// TIA Portal V20 export
FUNCTION "Service_Dosing" : Void   // FC11, FBD
TITLE = Service
{ S7_Optimized_Access := 'TRUE' }
AUTHOR : Siemens AG
FAMILY : ServiceControl
VERSION : 1.0
// stored: SetENOAutomatically false
   VAR_TEMP
      State : "Service_States";
   END_VAR
BEGIN

REGION Network 1: Cm P100 feedback
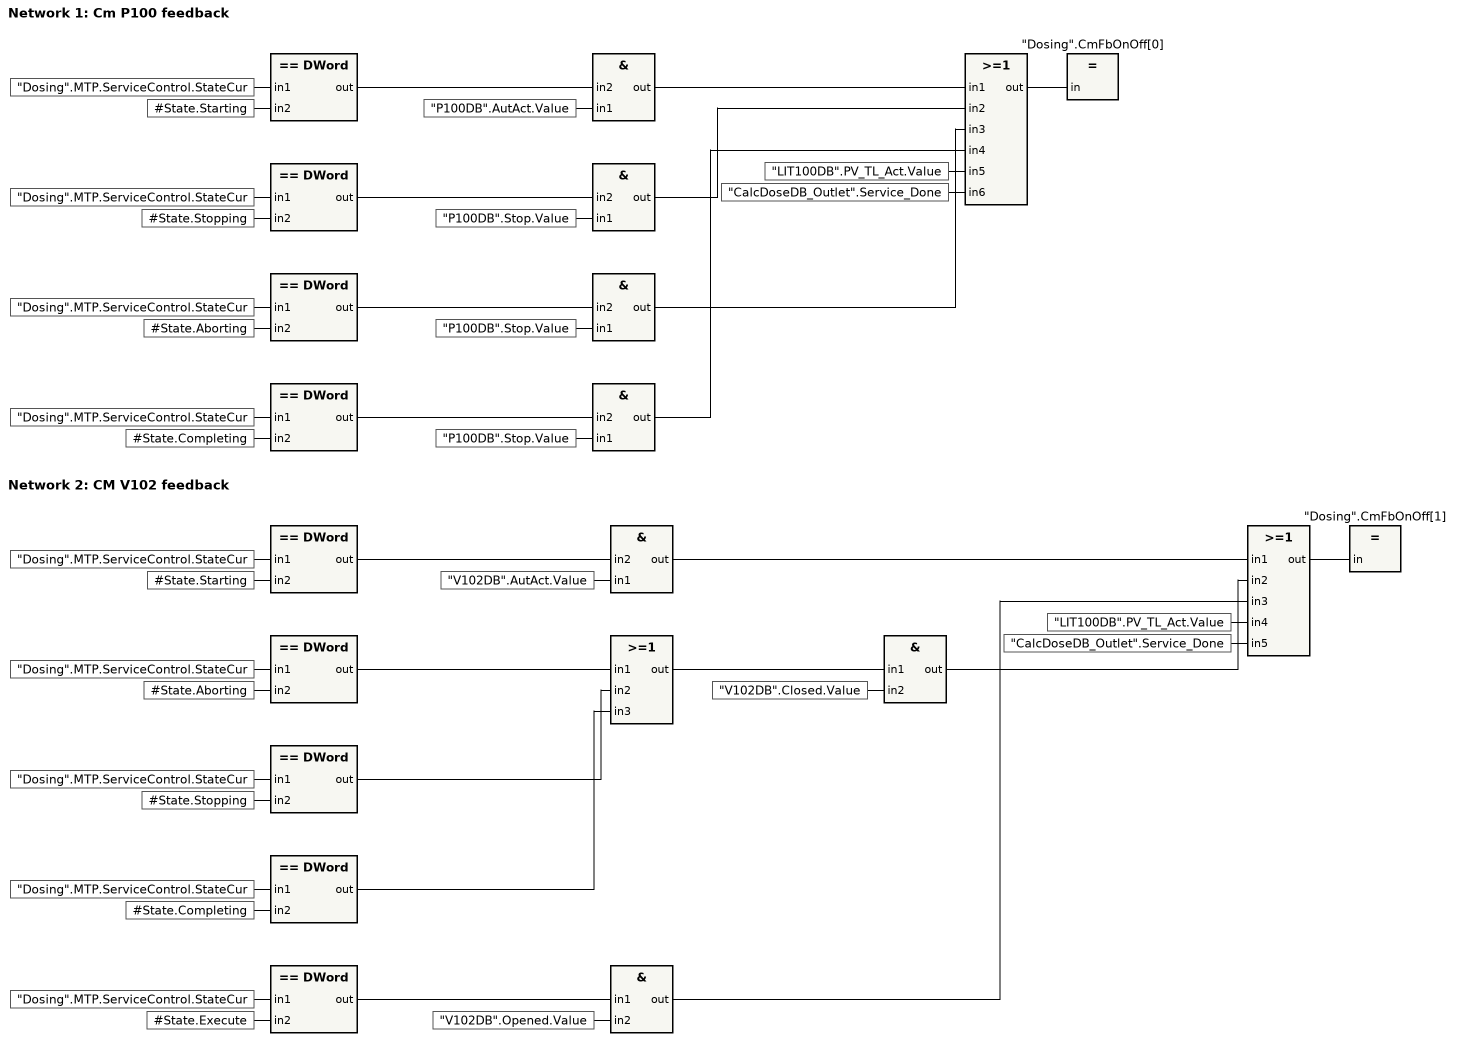
   "Dosing".CmFbOnOff[0] := (("Dosing".MTP.ServiceControl.StateCur = #State.Starting) AND "P100DB".AutAct.Value) OR (("Dosing".MTP.ServiceControl.StateCur = #State.Stopping) AND "P100DB".Stop.Value) OR (("Dosing".MTP.ServiceControl.StateCur = #State.Aborting) AND "P100DB".Stop.Value) OR (("Dosing".MTP.ServiceControl.StateCur = #State.Completing) AND "P100DB".Stop.Value) OR "LIT100DB".PV_TL_Act.Value OR "CalcDoseDB_Outlet".Service_Done;
END_REGION

REGION Network 2: CM V102 feedback
   "Dosing".CmFbOnOff[1] := (("Dosing".MTP.ServiceControl.StateCur = #State.Starting) AND "V102DB".AutAct.Value) OR ((("Dosing".MTP.ServiceControl.StateCur = #State.Aborting) OR ("Dosing".MTP.ServiceControl.StateCur = #State.Stopping) OR ("Dosing".MTP.ServiceControl.StateCur = #State.Completing)) AND "V102DB".Closed.Value) OR (("Dosing".MTP.ServiceControl.StateCur = #State.Execute) AND "V102DB".Opened.Value) OR "LIT100DB".PV_TL_Act.Value OR "CalcDoseDB_Outlet".Service_Done;
END_REGION

REGION Network 3: CM V103 feedback
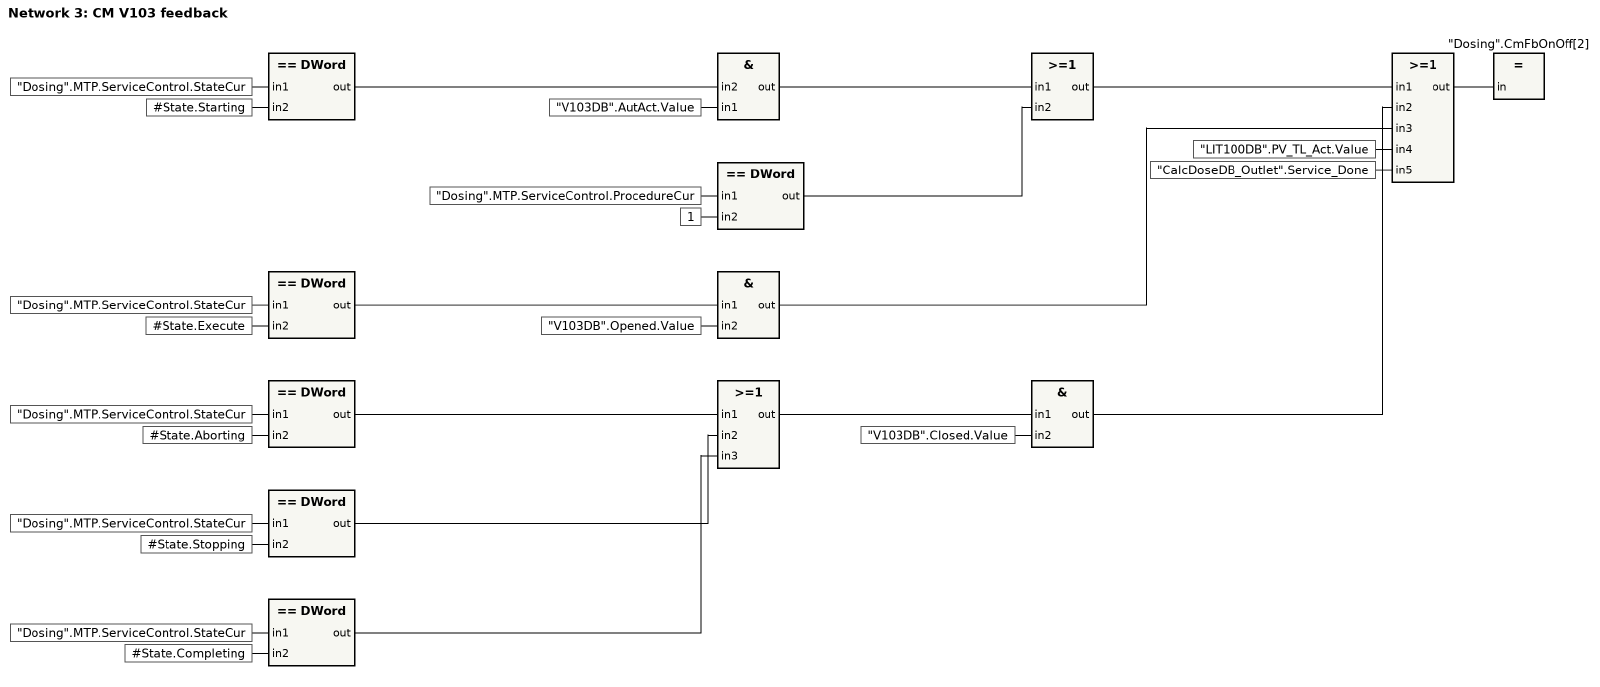
   "Dosing".CmFbOnOff[2] := (("Dosing".MTP.ServiceControl.StateCur = #State.Starting) AND "V103DB".AutAct.Value) OR ("Dosing".MTP.ServiceControl.ProcedureCur = 1) OR ((("Dosing".MTP.ServiceControl.StateCur = #State.Aborting) OR ("Dosing".MTP.ServiceControl.StateCur = #State.Stopping) OR ("Dosing".MTP.ServiceControl.StateCur = #State.Completing)) AND "V103DB".Closed.Value) OR (("Dosing".MTP.ServiceControl.StateCur = #State.Execute) AND "V103DB".Opened.Value) OR "LIT100DB".PV_TL_Act.Value OR "CalcDoseDB_Outlet".Service_Done;
END_REGION

REGION Network 4: CM V104 feedback
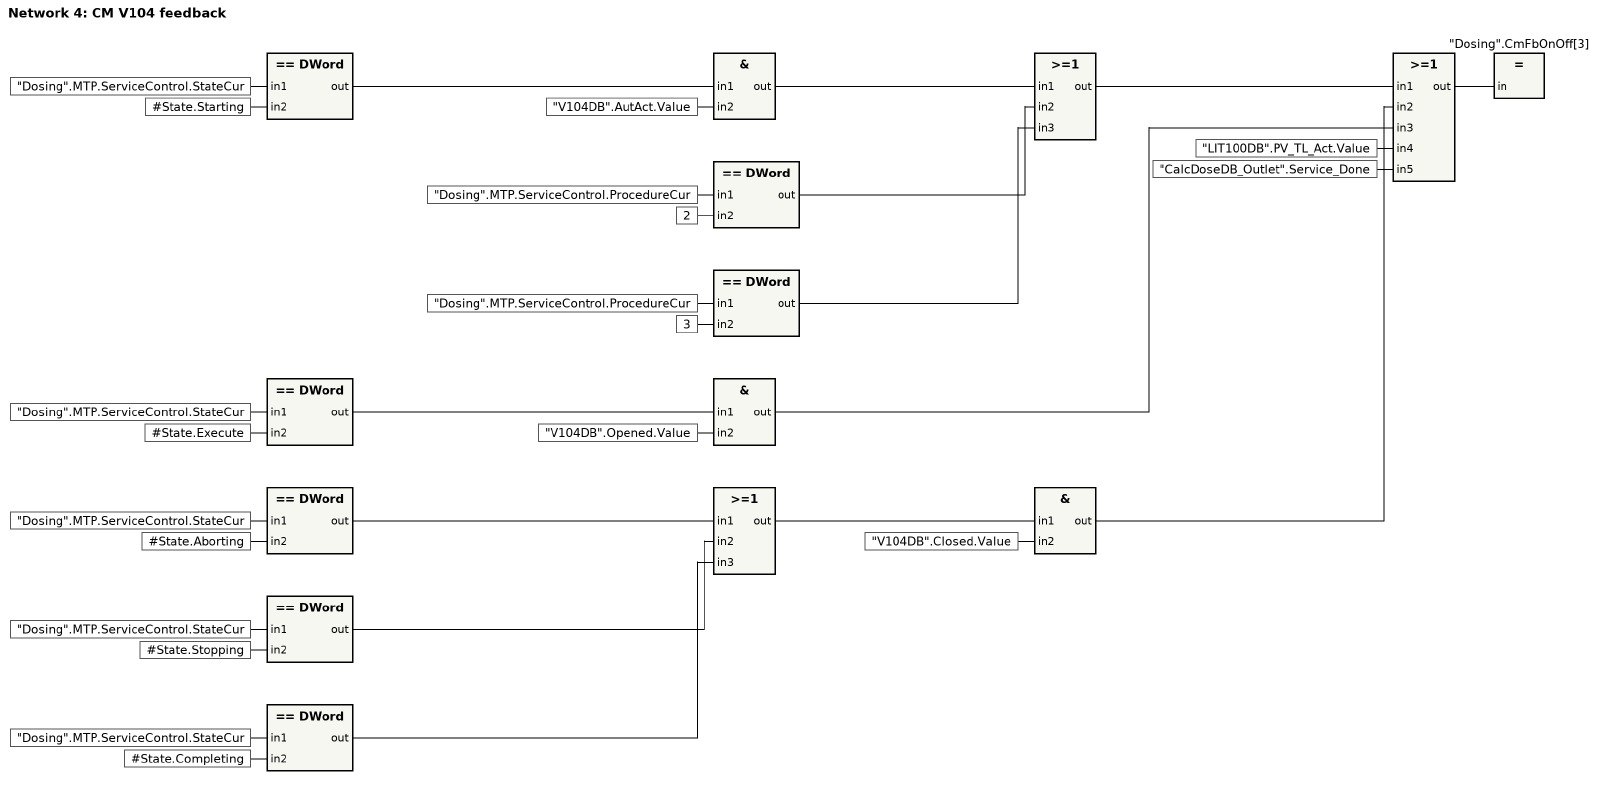
   "Dosing".CmFbOnOff[3] := (("Dosing".MTP.ServiceControl.StateCur = #State.Starting) AND "V104DB".AutAct.Value) OR ("Dosing".MTP.ServiceControl.ProcedureCur = 2) OR ("Dosing".MTP.ServiceControl.ProcedureCur = 3) OR ((("Dosing".MTP.ServiceControl.StateCur = #State.Aborting) OR ("Dosing".MTP.ServiceControl.StateCur = #State.Stopping) OR ("Dosing".MTP.ServiceControl.StateCur = #State.Completing)) AND "V104DB".Closed.Value) OR (("Dosing".MTP.ServiceControl.StateCur = #State.Execute) AND "V104DB".Opened.Value) OR "LIT100DB".PV_TL_Act.Value OR "CalcDoseDB_Outlet".Service_Done;
END_REGION

REGION Network 5: Service
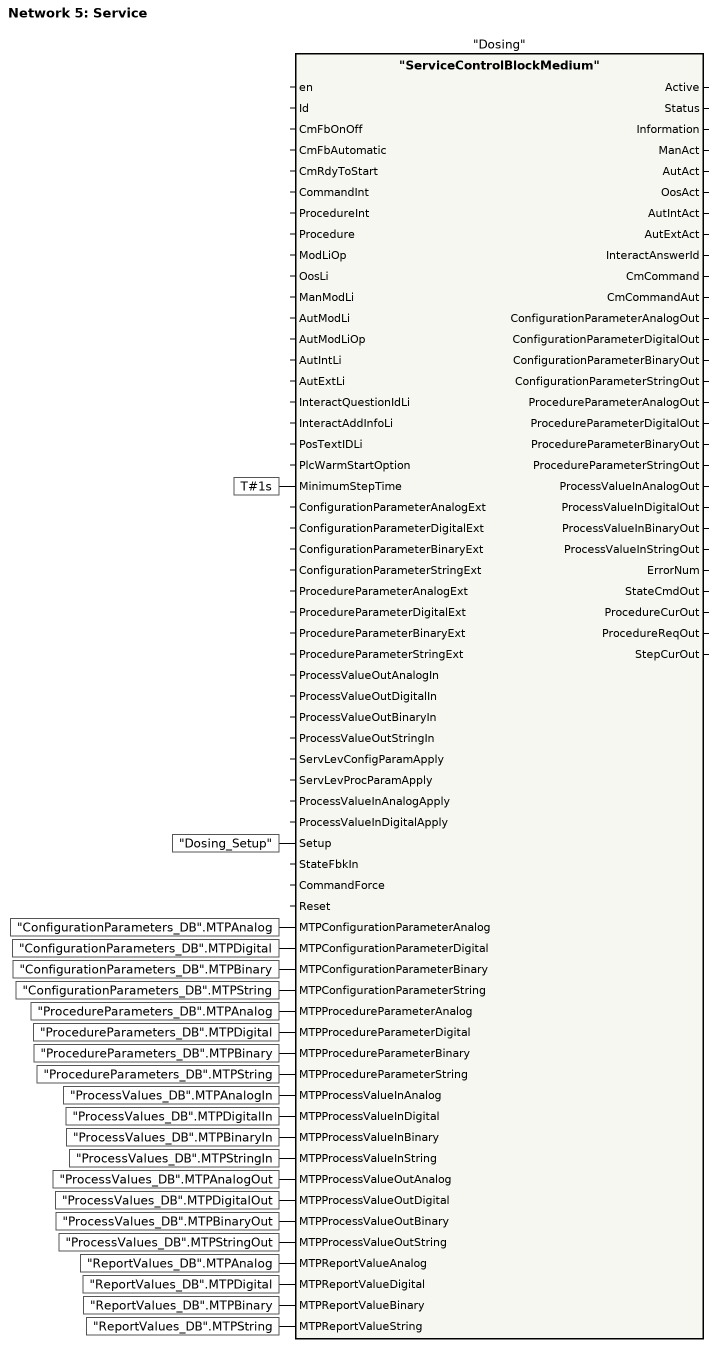
   "Dosing"(MinimumStepTime := T#1s,   // "ServiceControlBlockMedium"
            Setup := "Dosing_Setup",
            MTPConfigurationParameterAnalog := "ConfigurationParameters_DB".MTPAnalog,
            MTPConfigurationParameterDigital := "ConfigurationParameters_DB".MTPDigital,
            MTPConfigurationParameterBinary := "ConfigurationParameters_DB".MTPBinary,
            MTPConfigurationParameterString := "ConfigurationParameters_DB".MTPString,
            MTPProcedureParameterAnalog := "ProcedureParameters_DB".MTPAnalog,
            MTPProcedureParameterDigital := "ProcedureParameters_DB".MTPDigital,
            MTPProcedureParameterBinary := "ProcedureParameters_DB".MTPBinary,
            MTPProcedureParameterString := "ProcedureParameters_DB".MTPString,
            MTPProcessValueInAnalog := "ProcessValues_DB".MTPAnalogIn,
            MTPProcessValueInDigital := "ProcessValues_DB".MTPDigitalIn,
            MTPProcessValueInBinary := "ProcessValues_DB".MTPBinaryIn,
            MTPProcessValueInString := "ProcessValues_DB".MTPStringIn,
            MTPProcessValueOutAnalog := "ProcessValues_DB".MTPAnalogOut,
            MTPProcessValueOutDigital := "ProcessValues_DB".MTPDigitalOut,
            MTPProcessValueOutBinary := "ProcessValues_DB".MTPBinaryOut,
            MTPProcessValueOutString := "ProcessValues_DB".MTPStringOut,
            MTPReportValueAnalog := "ReportValues_DB".MTPAnalog,
            MTPReportValueDigital := "ReportValues_DB".MTPDigital,
            MTPReportValueBinary := "ReportValues_DB".MTPBinary,
            MTPReportValueString := "ReportValues_DB".MTPString);
END_REGION

REGION Network 6: Service HMI
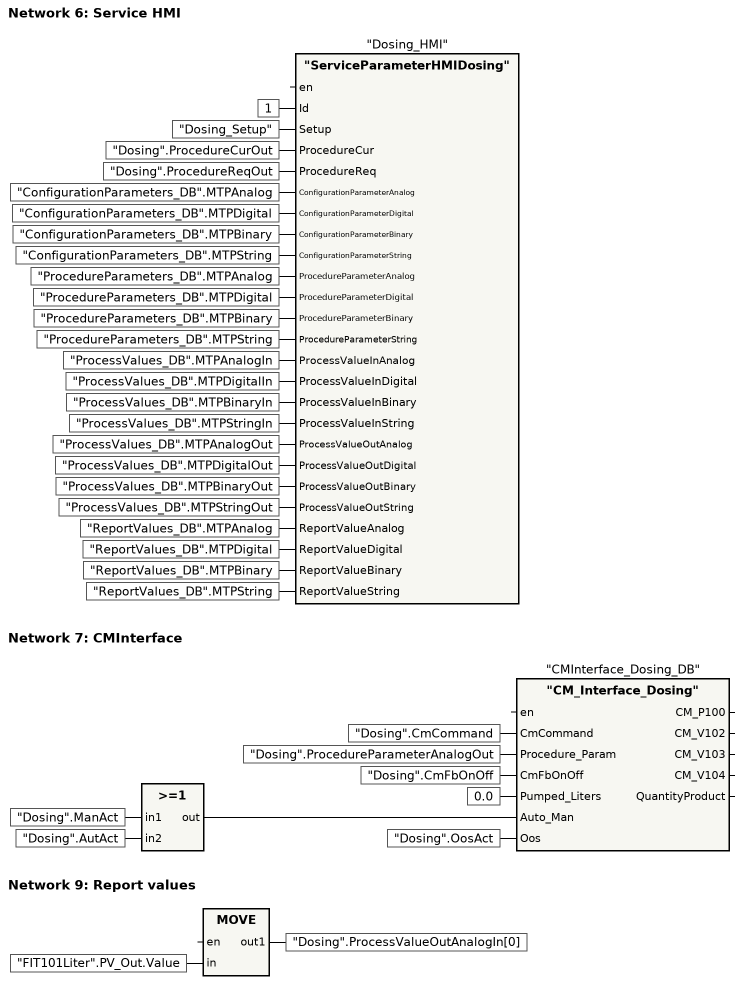
   "Dosing_HMI"(Id := 1,   // "ServiceParameterHMIDosing"
                Setup := "Dosing_Setup",
                ProcedureCur := "Dosing".ProcedureCurOut,
                ProcedureReq := "Dosing".ProcedureReqOut,
                ConfigurationParameterAnalog := "ConfigurationParameters_DB".MTPAnalog,
                ConfigurationParameterDigital := "ConfigurationParameters_DB".MTPDigital,
                ConfigurationParameterBinary := "ConfigurationParameters_DB".MTPBinary,
                ConfigurationParameterString := "ConfigurationParameters_DB".MTPString,
                ProcedureParameterAnalog := "ProcedureParameters_DB".MTPAnalog,
                ProcedureParameterDigital := "ProcedureParameters_DB".MTPDigital,
                ProcedureParameterBinary := "ProcedureParameters_DB".MTPBinary,
                ProcedureParameterString := "ProcedureParameters_DB".MTPString,
                ProcessValueInAnalog := "ProcessValues_DB".MTPAnalogIn,
                ProcessValueInDigital := "ProcessValues_DB".MTPDigitalIn,
                ProcessValueInBinary := "ProcessValues_DB".MTPBinaryIn,
                ProcessValueInString := "ProcessValues_DB".MTPStringIn,
                ProcessValueOutAnalog := "ProcessValues_DB".MTPAnalogOut,
                ProcessValueOutDigital := "ProcessValues_DB".MTPDigitalOut,
                ProcessValueOutBinary := "ProcessValues_DB".MTPBinaryOut,
                ProcessValueOutString := "ProcessValues_DB".MTPStringOut,
                ReportValueAnalog := "ReportValues_DB".MTPAnalog,
                ReportValueDigital := "ReportValues_DB".MTPDigital,
                ReportValueBinary := "ReportValues_DB".MTPBinary,
                ReportValueString := "ReportValues_DB".MTPString);
END_REGION

REGION Network 7: CMInterface
   "CMInterface_Dosing_DB"(CmCommand := "Dosing".CmCommand,   // "CM_Interface_Dosing"
                           Procedure_Param := "Dosing".ProcedureParameterAnalogOut,
                           CmFbOnOff := "Dosing".CmFbOnOff,
                           Pumped_Liters := 0.0,
                           Auto_Man := "Dosing".ManAct OR "Dosing".AutAct,
                           Oos := "Dosing".OosAct);
END_REGION

REGION Network 8: Block pause and hold state
END_REGION

REGION Network 9: Report values
   "Dosing".ProcessValueOutAnalogIn[0] := "FIT101Liter".PV_Out.Value;
END_REGION
END_FUNCTION
